PROGRAM MAIN
VAR
	fbTrig_Test				:BFB_Trigger;
	bTest					:BOOL;
	i						:INT;
	j						:INT;
END_VAR

fbTrig_Test(bIn := bTest);

IF fbTrig_Test.bRiseTrig THEN
	i := i + 1;
ELSIF fbTrig_Test.bFallTrig THEN
	i := i - 1;
END_IF

IF fbTrig_Test.bTrig THEN
	j := j + 1;
END_IF

END_PROGRAM

(* stored: Version 1.1.0.1, ProductVersion 3.1.4024.9
   POU MAIN: Id {5b321eb8-c770-40bd-8492-e3a6647735c9}, SpecialFunc None *)
